{attribute 'qualified_only'}
{attribute 'strict'}
TYPE E_TCPState :
(
	enum_member := 0
);
END_TYPE

(* stored: Version 1.1.0.1, ProductVersion 3.1.4024.12
   EnumerationTextList E_TCPState: Id {ed1492c9-7246-41ec-b3af-baa9c8a1f34f} *)
